TYPE St_RS232Word :
STRUCT
	inLength			: INT;
	overrunError		: BOOL;
	framingError		: BOOL;
	parityError 		: BOOL;
	bufferFull			: BOOL;
	initAccepted		: BOOL;
	recieveAccepted		: BOOL;
	transmitAccepted	: BOOL;
END_STRUCT
END_TYPE

(* stored: Version 1.1.0.1, ProductVersion 3.1.4024.9
   DUT St_RS232Word: Id {6b49e83d-7a56-4fcf-bec2-1434ff660cff} *)
